{attribute 'GeneratedUsingTerminal: KL9976-0050'}
{attribute addProperty BoxType "KL9976-0050"}
{attribute addProperty Id "Channel_1AT %I*0"}
{attribute addProperty CRC "1580138863"}
{attribute addProperty Size "0"}
TYPE KL_5E2F016F :
STRUCT
	{attribute addProperty Name "Channel_1"}
	Channel_1 : ;
END_STRUCT
END_TYPE

(* stored: Version 1.2.0.0, ProductVersion 3.1.4024.9
   DUT KL_5E2F016F: Id {ad539f16-29a5-406d-94fb-47d8737b6e9f} *)
